{attribute 'qualified_only'}
//{attribute 'strict'}
TYPE E_Pistons :
    (
        //Noon             := -1,
        LoadingBoxRegion := 0,
        ReturnRegion     := 1,
        AllocatedRegion  := 2

    )UINT;
END_TYPE

(* stored: Version 1.1.0.1, ProductVersion 3.1.4024.13
   DUT E_Pistons: Id {9bfafdba-d58e-4e93-812c-02fc65d7e8b3} *)
